				ELSIF stCycleDataNest1.bFail AND stCycleDataNest2.bFail THEN
					
					IF ctuRejectPart.CV > 1 AND NOT bPartPresentNest1 AND NOT bPartPresentNest2 THEN
						
						(* Renan Added 10Jul26 - Puck Locker *)
						IF bPuckLockerEnable THEN
							GVL_Stations.stPuckLocker.nRequestedRelease 		:= USINT#0;
							GVL_Stations.stPuckLocker.bApplyDisposition 		:= TRUE;
						END_IF
						(*\Renan Added 10Jul26 - Puck Locker *)
						
						eCycleState												:= E_General_ProcessCycle.NEST_CLEARING;
					
					ELSIF ctuRejectPart.CV > 1 AND ( bPartPresentNest1 OR bPartPresentNest2) THEN
						
						bRejectPartFault										:= TRUE; 		
					
					END_IF;
					
					sMachineMessage												:= 'REMOVE PART FROM BOTH NESTS AND PUT IN REJECT CHUTE';
					
				END_IF
				
E_General_ProcessCycle.NEST_CLEARING:

				stCamera.CMD.CameraCMD.ContinuousPartPresent1					:= bProcessedPart[0];
				stCamera.CMD.CameraCMD.ContinuousPartPresent2					:= bProcessedPart[1];
				stCamera.CMD.bExecute											:= TRUE;
				
				IF bPuckLockerEnable AND GVL_Stations.stPuckLocker.eState = E_PuckLockerState.WaitingForNestsEmpty THEN
				
					IF (bPartPresentNest1 AND bNest1Flag) OR (bPartPresentNest2 AND bNest2Flag) THEN
						
						sMachineMessage 										:= 'Remove parts from nests to release puck';
						
					ELSE
						
						sMachineMessage 										:= 'Waiting for puck to be released';
						
					END_IF
				
				ELSIF (bPartPresentNest1 AND bNest1Flag) AND NOT (bPartPresentNest2 AND bNest2Flag)  THEN
					
					IF bPuckLockerEnable THEN
						
						sMachineMessage 										:= 'Remove processed part from nest 1 to release puck';
						
					ELSE
						
						sMachineMessage 										:= 'Remove Processed part from nest 1';
						
					END_IF
					
				ELSIF NOT (bPartPresentNest1 AND bNest1Flag) AND (bPartPresentNest2 AND bNest2Flag)  THEN 
					
					IF bPuckLockerEnable THEN
						
						sMachineMessage 										:= 'Remove processed part from nest 2 to release puck';
						
					ELSE
						
						sMachineMessage 										:= 'Remove Processed part from nest 2';
						
					END_IF
					
				ELSIF (bPartPresentNest1 AND bNest1Flag) AND (bPartPresentNest2 AND bNest2Flag) THEN 
					
					IF bPuckLockerEnable THEN
						
						sMachineMessage 										:= 'Remove processed parts to release puck';
						
					ELSE
						
						sMachineMessage 										:= 'Remove Processed parts';
						
					END_IF
					
				ELSIF (NOT bPartPresentNest1 OR NOT bNest1Flag) AND (NOT bPartPresentNest2 OR NOT bNest2Flag)  THEN
					
					sMachineMessage 											:= '';
					eCycleState													:= E_General_ProcessCycle.RESET_ALL_CMD;
									
				END_IF
			
				
END_CASE
END_ACTION

ACTION c_ACT_SaveData:

//SAVING NEST 1 DATA

IF bProcessedPart[0] THEN
		
	IF stCycleDataNest1.bPass THEN
	
		stCycleDataNest1.sGeneralResult			:= 'PASS';

	ELSIF stCycleDataNest1.bFail THEN
	
		stCycleDataNest1.sGeneralResult			:= 'FAIL';

	END_IF

	IF stCycleDataNest1.LSS_Pass THEN
	
		stCycleDataNest1.sHeightTestResult		:= 'PASS';
	
	ELSIF stCycleDataNest1.LSS_Fail THEN
	
		stCycleDataNest1.sHeightTestResult		:= 'FAIL';
	
	END_IF



	IF stCycleDataNest1.LeakTest_Pass THEN
	
		stCycleDataNest1.sLeakTesterResult		:= 'PASS';

	ELSIF stCycleDataNest1.LeakTest_Fail THEN
	
		stCycleDataNest1.sLeakTesterResult		:= 'FAIL';
	
	END_IF
	
	stCycleDataNest1.sDistance1						:= REAL_TO_STRING(stCycleDataNest1.LSS_ScaledHeight[1]);
	stCycleDataNest1.sDistance2						:= REAL_TO_STRING(stCycleDataNest1.LSS_ScaledHeight[2]);
	stCycleDataNest1.sDistance3						:= REAL_TO_STRING(stCycleDataNest1.LSS_ScaledHeight[3]);
	stCycleDataNest1.sDistance4						:= REAL_TO_STRING(stCycleDataNest1.LSS_ScaledHeight[4]);
	
	stCycleDataNest1.sSetpoint1						:= REAL_TO_STRING(nHeightSetPoint);
	stCycleDataNest1.sSetpoint2						:= REAL_TO_STRING(nHeightSetPoint);
	stCycleDataNest1.sSetpoint3						:= REAL_TO_STRING(nHeightSetPoint);
	stCycleDataNest1.sSetpoint4						:= REAL_TO_STRING(nHeightSetPoint);
	
	aDataHistoryNest1[0]						:= stCycleDataNest1;
	
END_IF
	

//SAVING NEST 2 DATA

IF bProcessedPart[1] THEN
	
	IF stCycleDataNest2.bPass THEN
	
		stCycleDataNest2.sGeneralResult			:= 'PASS';

	ELSIF stCycleDataNest2.bFail THEN
	
		stCycleDataNest2.sGeneralResult			:= 'FAIL';

	END_IF

	IF stCycleDataNest2.LSS_Pass THEN
	
		stCycleDataNest2.sHeightTestResult		:= 'PASS';
	
	ELSIF stCycleDataNest2.LSS_Fail THEN
	
		stCycleDataNest2.sHeightTestResult		:= 'FAIL';
	
	END_IF



	IF stCycleDataNest2.LeakTest_Pass THEN
	
		stCycleDataNest2.sLeakTesterResult		:= 'PASS';

	ELSIF stCycleDataNest2.LeakTest_Fail THEN
	
		stCycleDataNest2.sLeakTesterResult		:= 'FAIL';
	
	END_IF
	
	stCycleDataNest2.sDistance1						:= REAL_TO_STRING(stCycleDataNest2.LSS_ScaledHeight[1]);
	stCycleDataNest2.sDistance2						:= REAL_TO_STRING(stCycleDataNest2.LSS_ScaledHeight[2]);
	stCycleDataNest2.sDistance3						:= REAL_TO_STRING(stCycleDataNest2.LSS_ScaledHeight[3]);
	stCycleDataNest2.sDistance4						:= REAL_TO_STRING(stCycleDataNest2.LSS_ScaledHeight[4]);
	
	stCycleDataNest2.sSetpoint1						:= REAL_TO_STRING(nHeightSetPoint);
	stCycleDataNest2.sSetpoint2						:= REAL_TO_STRING(nHeightSetPoint);
	stCycleDataNest2.sSetpoint3						:= REAL_TO_STRING(nHeightSetPoint);
	stCycleDataNest2.sSetpoint4						:= REAL_TO_STRING(nHeightSetPoint);
	
	aDataHistoryNest2[0]						:= stCycleDataNest2;
	
END_IF
END_ACTION

ACTION d_ACT_IO:
//INPUTS

rRejectSensor( CLK := dw_T08_EL1809.iRejectSensor);

bDoorClosingFlag					:= (eCycleState = E_General_ProcessCycle.CLOSE_PROCESS_DOOR) OR (eCycleState = E_General_ProcessCycle.WAIT_CLOSE_PROCESS_DOOR) OR 
										bDoorClosingInitFlag;
bDoorOpeningFlag					:= eCycleState = E_General_ProcessCycle.OPEN_PROCESS_DOOR;

bProcessDoorClosedConditionFlag		:=  eCycleState = E_General_ProcessCycle.EXTEND_PROCESS_CYLINDER OR
										eCycleState = E_General_ProcessCycle.WAIT_EXTEND_PROCESS_CYLINDER OR
										eCycleState = E_General_ProcessCycle.RETRACT_PROCESS_CYLINDER OR
										eCycleState = E_General_ProcessCycle.WAIT_RETRACT_PROCESS_CYLINDER OR
										eCycleState = E_General_ProcessCycle.HOLD_PART OR
										eCycleState = E_General_ProcessCycle.WAIT_HOLD_PART OR
										eCycleState = E_General_ProcessCycle.RELEASE_PART OR
										eCycleState = E_General_ProcessCycle.WAIT_RELEASE_PART OR
										eCycleState = E_General_ProcessCycle.VACUUM_CYLINDER_EXTENSION OR
										eCycleState = E_General_ProcessCycle.WAIT_VACUUM_CYLINDER_EXTENSION OR
										eCycleState = E_General_ProcessCycle.VACUUM_CYLINDER_RETRACTION OR
										eCycleState = E_General_ProcessCycle.WAIT_VACUUM_CYLINDER_RETRACTION;
					

										

										
tonTwoHandsSignal( IN := stTwinSAFE.qTwoHandsSafe , PT := stTimers.tTwoHandsSignal);						
				
bTwoHandsSignal						:= tonTwoHandsSignal.Q;
		
dw_T09_EL2809.qIndicatorLED1_Red	:= stCycleDataNest1.bFail;		
dw_T09_EL2809.qIndicatorLED1_Green	:= stCycleDataNest1.bPass;	
dw_T09_EL2809.qIndicatorLED2_Red	:= stCycleDataNest2.bFail;		
dw_T09_EL2809.qIndicatorLED2_Green	:= stCycleDataNest2.bPass;	

bPartPresent[0]					:= 	bProcessedPart[0];
bPartPresent[1]					:= 	bProcessedPart[1];
	

				
stTwinSAFE.iMachineHoming_Manual		:= 	stMachineStatus.eMachineState = E_MachineState.SAFETY OR
										stMachineStatus.eMachineState = E_MachineState.SYSTEM_INITIALISING OR 
										stMachineStatus.eMachineState = E_MachineState.MANUAL_MODE;												
										
//General Stations CMD
	
stVacuumCylinder.CMD.bAbort			:= bGeneralAbort;
stCamera.CMD.bAbort					:= bGeneralAbort;	
stLeakTesters.CMD.bAbort			:= bGeneralAbort;	
stLSS.CMD.bAbort					:= bGeneralAbort;
stProcessCylinder.CMD.bAbort		:= bGeneralAbort;
stProcessDoor.CMD.bAbort			:= bGeneralAbort;

stVacuumCylinder.CMD.bEnable		:= bGeneralEnable;
stCamera.CMD.bEnable				:= bGeneralEnable;	
stLeakTesters.CMD.bEnable			:= bGeneralEnable;	
stLSS.CMD.bEnable					:= bGeneralEnable;
stProcessCylinder.CMD.bEnable		:= bGeneralEnable;
stProcessDoor.CMD.bEnable			:= bGeneralEnable;

stVacuumCylinder.CMD.bReset			:= bGeneralRST;
stCamera.CMD.bReset					:= bGeneralRST;	
stLeakTesters.CMD.bReset			:= bGeneralRST;	
stLSS.CMD.bReset					:= bGeneralRST;
stProcessCylinder.CMD.bReset		:= bGeneralRST;
stProcessDoor.CMD.bReset			:= bGeneralRST;

stVacuumCylinder.CMD.bManualMode	:= bGeneralManualMode;
stCamera.CMD.bManualMode			:= bGeneralManualMode;
stLeakTesters.CMD.bManualMode		:= bGeneralManualMode;
stLSS.CMD.bManualMode				:= bGeneralManualMode;
stProcessCylinder.CMD.bManualMode	:= bGeneralManualMode;
stProcessDoor.CMD.bManualMode		:= bGeneralManualMode;
END_ACTION

END_PROGRAM

// ---- POUs/B_STATIONS/B_5_PUCK_LOCKER/B_5_1_PRG_PuckLocker.TcPOU
PROGRAM B_5_1_PRG_PuckLocker
VAR
	// ============================================================
    // Local process variables
    // ============================================================
    eMode                       : E_PuckLockerMode;

    bPuckPresentRaw             : BOOL;
    bPuckPresent                : BOOL;

    bPuckSensorsMismatchRaw     : BOOL;
    bPuckSensorsMismatch        : BOOL;

    bEnableEmptyPuckBypass      : BOOL;


    // ============================================================
    // Edge detection
    // ============================================================
    rTrigPuckPresent          : R_TRIG;
    fTrigPuckPresent          : F_TRIG;

    rTrigApplyDisposition     : R_TRIG;
    rTrigEmptyPuckBypass      : R_TRIG;
    rTrigAcknowledgeFault     : R_TRIG;


    // ============================================================
    // Timers
    // ============================================================
    tonPuckPresentOnDelay        : TON;
    tonPuckPresentOffDelay       : TON;

    tonPuckMismatchDelay         : TON;
	tonPuckPresentDebounce		 : TON;
	
    tonPinLockDelay              : TON;
	
END_VAR

// =================================================================
// 1. Engineering / HMI configuration
// =================================================================
// eMode should be persistent through your existing GVL_HMI Persistent
// implementation, or copied there from the Engineering page.
// =================================================================
// Puck locker HMI mode selection
// =================================================================


(* Renan Added 10Jul26 - Puck Locker common code *)


    IF NOT GVL_HMI.bPuckLockerGateEnable THEN
        GVL_HMI.bPuckLockerSkipEnable := FALSE;
    END_IF;

    IF NOT GVL_HMI.bPuckLockerGateEnable THEN

        eMode := E_PuckLockerMode.Disabled;

    ELSIF GVL_HMI.bPuckLockerSkipEnable THEN

        eMode := E_PuckLockerMode.EnabledWithEmptyPuckBypass;

    ELSE

        eMode := E_PuckLockerMode.Enabled;

    END_IF;

    GVL_HMI.ePuckLockerMode := eMode;
    GVL_HMI.stPuckLocker.eMode := eMode;


(*\Renan Added 10Jul26 - Puck Locker common code *)

// Skip option is never allowed while gate is disabled.
IF NOT GVL_HMI.bPuckLockerGateEnable THEN
    GVL_HMI.bPuckLockerSkipEnable := FALSE;
END_IF;

// Convert HMI toggles into the internal locker mode.
IF NOT GVL_HMI.bPuckLockerGateEnable THEN

    eMode := E_PuckLockerMode.Disabled;

ELSIF GVL_HMI.bPuckLockerSkipEnable THEN

    eMode := E_PuckLockerMode.EnabledWithEmptyPuckBypass;

ELSE

    eMode := E_PuckLockerMode.Enabled;

END_IF;

// Keep existing status/interface compatible.
GVL_HMI.ePuckLockerMode := eMode;
GVL_HMI.stPuckLocker.eMode := eMode;


// =================================================================
// 2. Read physical inputs
// =================================================================
GVL_Stations.stPuckLocker.bPuckSensorUp 	:= GVL_IO.dw_T08_EL1809.iPuckSensorUp;
GVL_Stations.stPuckLocker.bPuckSensorDown 	:= GVL_IO.dw_T08_EL1809.iPuckSensorDown;

// =================================================================
// 3. Validate puck presence
// =================================================================
// The puck is considered correctly positioned only when both sensors
// are active simultaneously.
bPuckPresentRaw := GVL_Stations.stPuckLocker.bPuckSensorUp AND GVL_Stations.stPuckLocker.bPuckSensorDown;

GVL_IO.stTwinSAFE.iPuckError := GVL_Stations.stPuckLocker.bUnexpectedRemovalFault;

// One sensor ON and the other OFF may be caused by:
// - puck moving through the sensing area;
// - puck not aligned;
// - puck partially lifted;
// - sensor issue.
bPuckSensorsMismatchRaw :=GVL_Stations.stPuckLocker.bPuckSensorUp XOR GVL_Stations.stPuckLocker.bPuckSensorDown;

// Require both sensors active for 100 ms before confirming puck.
tonPuckPresentOnDelay(IN := bPuckPresentRaw,PT := T#100MS);

// Require both sensors inactive for 100 ms before confirming absence.
tonPuckPresentOffDelay(IN := NOT bPuckPresentRaw,PT := T#100MS);


IF tonPuckPresentOnDelay.Q THEN

    bPuckPresent := TRUE;

ELSIF tonPuckPresentOffDelay.Q THEN

    bPuckPresent := FALSE;

END_IF

// Debounce puck present
tonPuckPresentDebounce(IN := bPuckPresentRaw, PT := T#100MS);

// Debounced puck detection
GVL_Stations.stPuckLocker.bPuckDetected := tonPuckPresentDebounce.Q;

// Keep mismatch indication only after a short delay, so normal puck
// movement does not generate false warnings.
tonPuckMismatchDelay(IN := bPuckSensorsMismatchRaw,PT := T#500MS);

bPuckSensorsMismatch := tonPuckMismatchDelay.Q;

// =================================================================
// 4. Edge detection
// =================================================================
rTrigPuckPresent(CLK := bPuckPresent);

fTrigPuckPresent(CLK := bPuckPresent);

rTrigApplyDisposition(CLK := GVL_Stations.stPuckLocker.bApplyDisposition);

rTrigEmptyPuckBypass(CLK := GVL_HMI.stPuckLocker.bCmdEmptyPuckBypass);

rTrigAcknowledgeFault(CLK := GVL_HMI.stPuckLocker.bCmdAcknowledgeRemovalFault);


// =================================================================
// 5. Latch disposition request from MachineCtrl
// =================================================================
// MachineCtrl should write these values once, after both final nest
// results are known:
//
// PASS / PASS:
// nRequestedRelease := 2;
// nRequestedRemoval := 0;
//
// PASS / FAIL or FAIL / PASS:
// nRequestedRelease := 1;
// nRequestedRemoval := 0;
//
// FAIL / FAIL:
// nRequestedRelease := 0;
// nRequestedRemoval := 1;
//
// bApplyDisposition := TRUE;
IF rTrigApplyDisposition.Q THEN

    IF GVL_Stations.stPuckLocker.nRequestedRelease > USINT#2 THEN
        GVL_Stations.stPuckLocker.nPucksAllowedToPass := USINT#2;
    ELSE
        GVL_Stations.stPuckLocker.nPucksAllowedToPass :=
            GVL_Stations.stPuckLocker.nRequestedRelease;
    END_IF

    GVL_Stations.stPuckLocker.bDispositionPending := TRUE;
    GVL_Stations.stPuckLocker.bApplyDisposition := FALSE;

END_IF


// =================================================================
// 6. Default values
// =================================================================
GVL_Stations.stPuckLocker.bRemovalAllowed := FALSE;
bEnableEmptyPuckBypass := FALSE;

tonPinLockDelay(IN := GVL_Stations.stPuckLocker.eState = E_PuckLockerState.LockingPuck AND bPuckPresent, PT := T#300MS);

IF stMachineStatus.bInitialising OR stMachineStatus.eMachineState = E_MachineState.SYSTEM_INITIALISING THEN

    f_ACT_ResetPuckLocker();
    RETURN;

END_IF

// =================================================================
// 8. Main Puck Locker State Machine
// =================================================================
CASE GVL_Stations.stPuckLocker.eState OF


    // ------------------------------------------------------------
    // Locker disabled.
    // Pin remains down and does not interfere with puck movement.
    // ------------------------------------------------------------
    E_PuckLockerState.Disabled:

        GVL_Stations.stPuckLocker.bPinCommandUp := FALSE;

        GVL_Stations.stPuckLocker.bPuckLocked := FALSE;
        GVL_Stations.stPuckLocker.bUnexpectedRemovalFault := FALSE;

        GVL_Stations.stPuckLocker.nPucksAllowedToPass := 0;
        GVL_Stations.stPuckLocker.nPucksToRemove := 0;

        GVL_Stations.stPuckLocker.bDispositionPending := FALSE;
        GVL_Stations.stPuckLocker.bDispositionHandled := FALSE;

        IF eMode <> E_PuckLockerMode.Disabled THEN

            GVL_Stations.stPuckLocker.eState := E_PuckLockerState.WaitingForPuck;

        END_IF


    // ------------------------------------------------------------
    // Pin remains down. Wait for a properly centred puck.
    // ------------------------------------------------------------
    E_PuckLockerState.WaitingForPuck:

        GVL_Stations.stPuckLocker.bPinCommandUp := FALSE;
        GVL_Stations.stPuckLocker.bPuckLocked := FALSE;

        IF eMode = E_PuckLockerMode.Disabled THEN

            GVL_Stations.stPuckLocker.eState := E_PuckLockerState.Disabled;

        ELSIF bPuckPresent
              AND GVL_Stations.stPuckLocker.nPucksAllowedToPass = 0
              AND GVL_Stations.stPuckLocker.nPucksToRemove = 0 THEN

            GVL_Stations.stPuckLocker.eState := E_PuckLockerState.LockingPuck;

        END_IF


    // ------------------------------------------------------------
    // Pin command is up.
    // No physical feedback exists, so locking is accepted after
    // 300 ms while the puck stays detected.
    // ------------------------------------------------------------
    E_PuckLockerState.LockingPuck:

        GVL_Stations.stPuckLocker.bPinCommandUp := TRUE;
		GVL_Stations.stPuckLocker.bPuckLocked := FALSE;
	
		IF eMode = E_PuckLockerMode.Disabled THEN
	
			GVL_Stations.stPuckLocker.eState := E_PuckLockerState.Disabled;
	
		ELSIF NOT bPuckPresent THEN
	
			// Puck was not fully captured yet.
			// Return to waiting state without fault.
			GVL_Stations.stPuckLocker.eState := E_PuckLockerState.WaitingForPuck;
	
		ELSIF tonPinLockDelay.Q THEN
	
			GVL_Stations.stPuckLocker.bPuckLocked := TRUE;
			GVL_Stations.stPuckLocker.eState := E_PuckLockerState.Locked;
	
		END_IF


    // ------------------------------------------------------------
    // Puck captured by locker pin.
    // Wait for process disposition, bypass request or fault.
    // ------------------------------------------------------------
    E_PuckLockerState.Locked:

        GVL_Stations.stPuckLocker.bPinCommandUp := TRUE;
        GVL_Stations.stPuckLocker.bPuckLocked := TRUE;


        // Bypass is only allowed in the configured bypass mode.
        // It is disabled once a process disposition is pending.
        bEnableEmptyPuckBypass := (eMode = E_PuckLockerMode.EnabledWithEmptyPuckBypass) AND NOT GVL_Stations.stPuckLocker.bDispositionPending AND NOT GVL_Stations.stPuckLocker.bUnexpectedRemovalFault;


        // Puck disappeared while pin should have been holding it.
        IF NOT bPuckPresent THEN

            GVL_Stations.stPuckLocker.bUnexpectedRemovalFault := TRUE;
            GVL_Stations.stPuckLocker.eState := E_PuckLockerState.UnexpectedPuckRemovalFault;


        // Empty puck bypass confirmed through HMI.
        ELSIF rTrigEmptyPuckBypass.Q
              AND bEnableEmptyPuckBypass THEN

            GVL_Stations.stPuckLocker.nPucksAllowedToPass := 1;
            GVL_Stations.stPuckLocker.nPucksToRemove := 0;

            GVL_HMI.stPuckLocker.bCmdEmptyPuckBypass := FALSE;

            GVL_Stations.stPuckLocker.eState := E_PuckLockerState.ReleasingPucks;


        // Final disposition received from MachineCtrl.
		ELSIF GVL_Stations.stPuckLocker.bDispositionPending THEN

			GVL_Stations.stPuckLocker.bDispositionPending := FALSE;
		
			// Release is authorised, but the pin must remain up until
			// both nests are empty. This ensures the PASS part was placed
			// back onto the locked puck before it can be released.
			IF GVL_Stations.stPuckLocker.nPucksAllowedToPass > 0 THEN
		
				GVL_Stations.stPuckLocker.eState := E_PuckLockerState.WaitingForNestsEmpty;
		
			END_IF
		END_IF


    E_PuckLockerState.WaitingForNestsEmpty:

		// Keep puck physically locked while either nest still contains
		// a product.
		GVL_Stations.stPuckLocker.bPinCommandUp := TRUE;
		GVL_Stations.stPuckLocker.bPuckLocked := TRUE;
	
		IF NOT bPuckPresent THEN
	
			GVL_Stations.stPuckLocker.bUnexpectedRemovalFault := TRUE;
	
			GVL_Stations.stPuckLocker.eState := E_PuckLockerState.UnexpectedPuckRemovalFault;
	
		ELSIF GVL_Stations.stPuckLocker.bNestsEmpty AND GVL_Stations.stPuckLocker.nPucksAllowedToPass > 0 THEN
	
			GVL_Stations.stPuckLocker.eState := E_PuckLockerState.ReleasingPucks;
	
		END_IF
		
    // ------------------------------------------------------------
    // Pin is down. One or two authorised pucks may pass.
    // A puck is counted when it clears both sensors.
    // ------------------------------------------------------------
    E_PuckLockerState.ReleasingPucks:

        GVL_Stations.stPuckLocker.bPinCommandUp := FALSE;
        GVL_Stations.stPuckLocker.bPuckLocked := FALSE;

        IF fTrigPuckPresent.Q
           AND GVL_Stations.stPuckLocker.nPucksAllowedToPass > 0 THEN

            GVL_Stations.stPuckLocker.nPucksAllowedToPass := GVL_Stations.stPuckLocker.nPucksAllowedToPass - 1;

        END_IF

        // All authorised pucks passed through the locker.
		// Return to rest/waiting state. No timeout is required here.
		IF GVL_Stations.stPuckLocker.nPucksAllowedToPass = 0
		AND NOT bPuckPresent THEN
		
			GVL_Stations.stPuckLocker.eState := E_PuckLockerState.WaitingForPuck;
		
		END_IF


    // ------------------------------------------------------------
    // Puck was removed unexpectedly while locked.
    // Pin stays down for safe recovery.
    //
    // Operator must return the puck to the sensor area and an
    // authorised user must acknowledge the event.
    // ------------------------------------------------------------
    E_PuckLockerState.UnexpectedPuckRemovalFault:

		GVL_Stations.stPuckLocker.bPinCommandUp := TRUE;
		GVL_Stations.stPuckLocker.bPuckLocked := FALSE;
	
		GVL_Stations.stPuckLocker.bUnexpectedRemovalFault := TRUE;
	
		IF eMode = E_PuckLockerMode.Disabled THEN
	
			GVL_Stations.stPuckLocker.eState := E_PuckLockerState.Disabled;
	
		ELSIF bPuckPresent AND rTrigAcknowledgeFault.Q THEN
		
			GVL_HMI.stPuckLocker.bCmdAcknowledgeRemovalFault := FALSE;
			GVL_Stations.stPuckLocker.bUnexpectedRemovalFault := FALSE;
			GVL_Stations.stPuckLocker.eState := E_PuckLockerState.LockingPuck;

		END_IF

END_CASE


// =================================================================
// 8. Write HMI interface
// =================================================================
GVL_HMI.stPuckLocker.bEnableEmptyPuckBypass := bEnableEmptyPuckBypass;

GVL_HMI.stPuckLocker.bPuckDetected := bPuckPresent;

GVL_HMI.stPuckLocker.bPuckLocked := GVL_Stations.stPuckLocker.bPuckLocked;

GVL_HMI.stPuckLocker.bPuckSensorMismatch := bPuckSensorsMismatch;

GVL_HMI.stPuckLocker.bUnexpectedRemovalFault := GVL_Stations.stPuckLocker.bUnexpectedRemovalFault;

GVL_HMI.stPuckLocker.bShowUnexpectedRemovalPopup := GVL_Stations.stPuckLocker.bUnexpectedRemovalFault;

GVL_HMI.stPuckLocker.nPucksAllowedToPass := GVL_Stations.stPuckLocker.nPucksAllowedToPass;


// This can remain FALSE if the HMI itself opens the confirmation
// popup after the operator presses the bypass button.
GVL_HMI.stPuckLocker.bShowEmptyPuckPopup := FALSE;



GVL_HMI.stPuckLocker.sMessage := GVL_Stations.stPuckLocker.sMessage;

// =================================================================
// 10. Physical output
// =================================================================
// This PRG must remain the only writer of the locker output.
GVL_IO.dw_T09_EL2809.qPuckLockerPinCommand := NOT GVL_Stations.stPuckLocker.bPinCommandUp;

ACTION f_ACT_ResetPuckLocker:
// ================================================================
// f_ACT_ResetPuckLocker
//
// Safe reset of puck locker internal state.
// Pin is commanded to release position.
// ================================================================

GVL_Stations.stPuckLocker.eState := E_PuckLockerState.WaitingForPuck;

GVL_Stations.stPuckLocker.bPinCommandUp := FALSE;
GVL_Stations.stPuckLocker.bPuckLocked := FALSE;
GVL_Stations.stPuckLocker.bRemovalAllowed := FALSE;

GVL_Stations.stPuckLocker.bUnexpectedRemovalFault := FALSE;

GVL_Stations.stPuckLocker.nPucksAllowedToPass := 0;
GVL_Stations.stPuckLocker.nPucksToRemove := 0;

GVL_Stations.stPuckLocker.nRequestedRelease := 0;
GVL_Stations.stPuckLocker.nRequestedRemoval := 0;

GVL_Stations.stPuckLocker.bApplyDisposition := FALSE;
GVL_Stations.stPuckLocker.bDispositionPending := FALSE;
GVL_Stations.stPuckLocker.bDispositionHandled := FALSE;

GVL_HMI.stPuckLocker.bCmdEmptyPuckBypass := FALSE;
GVL_HMI.stPuckLocker.bCmdAcknowledgeRemovalFault := FALSE;

GVL_HMI.stPuckLocker.bEnableEmptyPuckBypass := FALSE;
GVL_HMI.stPuckLocker.bShowUnexpectedRemovalPopup := FALSE;
GVL_HMI.stPuckLocker.bShowEmptyPuckPopup := FALSE;

GVL_HMI.stPuckLocker.bUnexpectedRemovalFault := FALSE;
GVL_HMI.stPuckLocker.nPucksAllowedToPass := 0;
GVL_HMI.stPuckLocker.sMessage := '';
END_ACTION

END_PROGRAM

// ---- POUs/D_CSV/D_1_PRG_CycleDataCSV.TcPOU
PROGRAM D_1_PRG_CycleDataCSV
VAR_INPUT
	
	stCycleDataNest1		: ST_CycleData;
	stCycleDataNest2		: ST_CycleData;
	bWriteNest1				: BOOL;
	bWriteNest2				: BOOL;
	
	
END_VAR
VAR_OUTPUT
	
	bCSVDone				: BOOL;
	bReady					: BOOL;
	
END_VAR
VAR
	sFileName		: T_MaxString := 'C:\Temp\USW_STN13_#date#.csv';(* CSV destination file path and name *)
	sCSVLine		: T_MaxString := '#1#;#2#;#3#;#4#;#5#;#6#;#7#;#8#;#9#,#10#,#11#,#12#,#13,#14,#15,#16,#17,#18#$L';
	bBusy			: BOOL;
	bError			: BOOL;
	nErrId			: UDINT;
	hFile			: UINT		:= 0;
	step			: DWORD 	:= 0;
	fbFileOpen		: FB_FileOpen;(* Opens file *)
	fbFileClose		: FB_FileClose;(* Closes file *)
	fbFilePuts		: FB_FilePuts;(* Writes one record (line) *)
	
	done: BOOL;
	
	f1_Nest			: STRING;
	f2_GeneralResult: STRING;
	f3_HeightResult	: STRING;
	f4_LeakTesterResult	: STRING;
	f5_Distance1	: STRING;
	f6_Distance2	: STRING;
	f7_Distance3	: STRING;
	f8_Distance4	: STRING;
	f9_Setpoint1	: STRING;
	f10_Setpoint2	: STRING;
	f11_Setpoint3	: STRING;
	f12_Setpoint4	: STRING;
	f13_RawValue1	: STRING;
	f14_RawValue2	: STRING;
	f15_RawValue3	: STRING;
	f16_RawValue4	: STRING;
	f17_Date		: STRING;
	f18_Time		: STRING;
	
	bWritingFirstRow : BOOL;
	bWrite			: BOOL;
	rWriteNest1		: R_TRIG;
	rWriteNest2		: R_TRIG;
	
	rError			: R_TRIG;
	
END_VAR



IF 	step = 0 THEN
	
		bReady		:= TRUE;

ELSE 	bReady		:= FALSE;
END_IF

CASE step OF
	0:	(* Wait for rising edge at bWrite variable *)
		bCSVDone	:= FALSE;
		IF bWrite	 THEN
			
			bWrite	:= FALSE;
			bBusy 	:= TRUE;
			bError	:= FALSE;
			nErrId	:= 0;
			hFile	:= 0;
			step 	:= 1;
			
		END_IF
		
	1:	(* Open source file *)
		fbFileOpen(  bExecute := FALSE  );
		fbFileOpen( sNetId := NetAmsIdLocal, 
					sPathName := sFileName, 
					nMode := FOPEN_MODEAPPEND OR FOPEN_MODETEXT,
					ePath := PATH_GENERIC, 
					bExecute := TRUE );
		step := 2;
	
	2:(* Wait until open not busy *)
		fbFileOpen( bExecute := FALSE, bError => bError, nErrID => nErrID, hFile => hFile );
		IF NOT fbFileOpen.bBusy THEN
			IF NOT fbFileOpen.bError THEN
				step := 3;
			ELSE(* Error: file not found? *)
				step := 100;
			END_IF
		END_IF

	3:(* Convert one PLC record to CSV format *)
		
		FindAndReplace(pSrcString:= ADR(sCSVLine), pDeleteString:= ADR('#1#'), pInsertString:= ADR(f1_Nest), pDstString:= ADR(sCSVLine), nDstSize:= SIZEOF(sCSVLine));
		FindAndReplace(pSrcString:= ADR(sCSVLine), pDeleteString:= ADR('#2#'), pInsertString:= ADR(f2_GeneralResult), pDstString:= ADR(sCSVLine), nDstSize:= SIZEOF(sCSVLine));
		FindAndReplace(pSrcString:= ADR(sCSVLine), pDeleteString:= ADR('#3#'), pInsertString:= ADR(f3_HeightResult), pDstString:= ADR(sCSVLine), nDstSize:= SIZEOF(sCSVLine));
		FindAndReplace(pSrcString:= ADR(sCSVLine), pDeleteString:= ADR('#4#'), pInsertString:= ADR(f4_LeakTesterResult), pDstString:= ADR(sCSVLine), nDstSize:= SIZEOF(sCSVLine));
		FindAndReplace(pSrcString:= ADR(sCSVLine), pDeleteString:= ADR('#5#'), pInsertString:= ADR(f5_Distance1), pDstString:= ADR(sCSVLine), nDstSize:= SIZEOF(sCSVLine));
		FindAndReplace(pSrcString:= ADR(sCSVLine), pDeleteString:= ADR('#6#'), pInsertString:= ADR(f6_Distance2), pDstString:= ADR(sCSVLine), nDstSize:= SIZEOF(sCSVLine));
		FindAndReplace(pSrcString:= ADR(sCSVLine), pDeleteString:= ADR('#7#'), pInsertString:= ADR(f7_Distance3), pDstString:= ADR(sCSVLine), nDstSize:= SIZEOF(sCSVLine));
		FindAndReplace(pSrcString:= ADR(sCSVLine), pDeleteString:= ADR('#8#'), pInsertString:= ADR(f8_Distance4), pDstString:= ADR(sCSVLine), nDstSize:= SIZEOF(sCSVLine));
		FindAndReplace(pSrcString:= ADR(sCSVLine), pDeleteString:= ADR('#9#'), pInsertString:= ADR(f9_Setpoint1), pDstString:= ADR(sCSVLine), nDstSize:= SIZEOF(sCSVLine));
		FindAndReplace(pSrcString:= ADR(sCSVLine), pDeleteString:= ADR('#10#'), pInsertString:= ADR(f10_Setpoint2), pDstString:= ADR(sCSVLine), nDstSize:= SIZEOF(sCSVLine));
		FindAndReplace(pSrcString:= ADR(sCSVLine), pDeleteString:= ADR('#11#'), pInsertString:= ADR(f11_Setpoint3), pDstString:= ADR(sCSVLine), nDstSize:= SIZEOF(sCSVLine));
		FindAndReplace(pSrcString:= ADR(sCSVLine), pDeleteString:= ADR('#12#'), pInsertString:= ADR(f12_Setpoint4), pDstString:= ADR(sCSVLine), nDstSize:= SIZEOF(sCSVLine));
		FindAndReplace(pSrcString:= ADR(sCSVLine), pDeleteString:= ADR('#13#'), pInsertString:= ADR(f13_RawValue1), pDstString:= ADR(sCSVLine), nDstSize:= SIZEOF(sCSVLine));
		FindAndReplace(pSrcString:= ADR(sCSVLine), pDeleteString:= ADR('#14#'), pInsertString:= ADR(f14_RawValue2), pDstString:= ADR(sCSVLine), nDstSize:= SIZEOF(sCSVLine));
		FindAndReplace(pSrcString:= ADR(sCSVLine), pDeleteString:= ADR('#15#'), pInsertString:= ADR(f15_RawValue3), pDstString:= ADR(sCSVLine), nDstSize:= SIZEOF(sCSVLine));
		FindAndReplace(pSrcString:= ADR(sCSVLine), pDeleteString:= ADR('#16#'), pInsertString:= ADR(f16_RawValue4), pDstString:= ADR(sCSVLine), nDstSize:= SIZEOF(sCSVLine));	
		FindAndReplace(pSrcString:= ADR(sCSVLine), pDeleteString:= ADR('#17#'), pInsertString:= ADR(f17_Date), pDstString:= ADR(sCSVLine), nDstSize:= SIZEOF(sCSVLine));
		FindAndReplace(pSrcString:= ADR(sCSVLine), pDeleteString:= ADR('#18#'), pInsertString:= ADR(f18_Time), pDstString:= ADR(sCSVLine), nDstSize:= SIZEOF(sCSVLine));
		done:=TRUE;
		
		IF done THEN
			step := 4;
			done := FALSE;
		ELSE
			step := 3;
		END_IF
		
		
	4:	(* Write single text line *)
		fbFilePuts( bExecute := FALSE );
		fbFilePuts( sNetId := '', 
					hFile := hFile, 
					sLine := sCSVLine, 
					bExecute := TRUE );
		step := 5;

	5:(* Wait until write not busy *)
		fbFilePuts( bExecute := FALSE, bError => bError, nErrID => nErrID );
		IF NOT fbFilePuts.bBusy THEN
			IF NOT fbFilePuts.bError THEN
				step := 10;
			ELSE(* Error *)
				step := 100;
			END_IF
		END_IF

	10:	(* Close source file *)
		fbFileClose( bExecute := FALSE );
		fbFileClose( sNetId := '', hFile := hFile, bExecute := TRUE );
		sCSVLine:= '#1#;#2#;#3#;#4#;#5#;#6#;#7#;#8#;#9#,#10#,#11#,#12#,#13#,#14#,#15#,#16#,#17#$L';
		step := 11;

	11:(* Wait until close not busy *)
		fbFileClose( bExecute := FALSE, bError => bError, nErrID => nErrID );
		IF ( NOT fbFileClose.bBusy ) THEN
			bWritingFirstRow	:= FALSE;
			
			hFile := 0;
			step := 100;
		END_IF

	100: (* Error or ready step => cleanup *)
		IF ( hFile <> 0 ) THEN
			step := 10; (* Close the source file *)
		ELSE
			bBusy := FALSE;
			step := 0;	(* Ready *)
			bCSVDone	:= TRUE;
		END_IF

END_CASE

IF (lastDateCSV <> sSystemDate) AND NOT (dw_T04_EL1918.iResetButton	OR stTester.bReset) THEN
lastDateCSV:= sSystemDate;
sFileName:= 'C:\Users\Administrator\Desktop\csv\CycleData_#date#.csv';
FindAndReplace(pSrcString:= ADR(sFileName), pDeleteString:= ADR('#date#'), pInsertString:= ADR(lastDateCSV), pDstString:= ADR(sFileName), nDstSize:= SIZEOF(sFileName));

f1_Nest			:= 'NEST';
f2_GeneralResult:= 'GENERAL RESULTS';
f3_HeightResult	:= 'HEIGHT CHECK RESULTS';
f4_LeakTesterResult	:= 'LEAK TESTER RESULTS';
f5_Distance1	:= 'DISTANCE 1';
f6_Distance2	:= 'DISTANCE 2';
f7_Distance3	:= 'DISTANCE 3';
f8_Distance4	:= 'DISTANCE 4';
f9_Setpoint1	:= 'SETPOINT 1';
f10_Setpoint2	:= 'SETPOINT 2';
f11_Setpoint3	:= 'SETPOINT 3';
f12_Setpoint4	:= 'SETPOINT 4';
f13_RawValue1	:= 'RAW HEIGHT 1';
f14_RawValue2	:= 'RAW HEIGHT 2';
f15_RawValue3	:= 'RAW HEIGHT 3';
f16_RawValue4	:= 'RAW HEIGHT 4';
f17_Date		:= 'DATE';
f18_Time		:= 'TIME';
bWrite			:= TRUE;
bWritingFirstRow	:= TRUE;

END_IF

IF NOT bWritingFirstRow THEN
	ACT_LinkingVariables();
END_IF

rError(CLK := bError);

bCSVError		:= rError.Q;

IF bWritingFirstRow AND (dw_T04_EL1918.iResetButton OR stTester.bReset) THEN
	
	lastDateCSV			:= '0';
	bCSVError			:= FALSE;			

END_IF

ACTION ACT_LinkingVariables:
rWriteNest1( CLK := bWriteNest1);
rWriteNest2( CLK := bWriteNest2);

IF rWriteNest1.Q THEN
	
	f1_Nest			:= INT_TO_STRING(stCycleDataNest1.nNest);
	f2_GeneralResult:= stCycleDataNest1.sGeneralResult;
	f3_HeightResult	:= stCycleDataNest1.sHeightTestResult;
	f4_LeakTesterResult	:= stCycleDataNest1.sLeakTesterResult;
	f5_Distance1	:= stCycleDataNest1.sDistance1;
	f6_Distance2	:= stCycleDataNest1.sDistance2;
	f7_Distance3	:= stCycleDataNest1.sDistance3;
	f8_Distance4	:= stCycleDataNest1.sDistance4;
	f9_Setpoint1	:= stCycleDataNest1.sSetpoint1;
	f10_Setpoint2	:= stCycleDataNest1.sSetpoint2;
	f11_Setpoint3	:= stCycleDataNest1.sSetpoint3;
	f12_Setpoint4	:= stCycleDataNest1.sSetpoint4;
	f13_RawValue1	:= REAL_TO_STRING(stCycleDataNest1.LSS_anRawMeasurement[1]);
	f14_RawValue2	:= REAL_TO_STRING(stCycleDataNest1.LSS_anRawMeasurement[2]);
	f15_RawValue3	:= REAL_TO_STRING(stCycleDataNest1.LSS_anRawMeasurement[3]);
	f16_RawValue4	:= REAL_TO_STRING(stCycleDataNest1.LSS_anRawMeasurement[4]);
	f17_Date		:= stCycleDataNest1.sDate;
	f18_Time		:= stCycleDataNest1.sTime;
	
	bWrite			:= TRUE;

ELSIF rWriteNest2.Q THEN
	
	f1_Nest			:= INT_TO_STRING(stCycleDataNest2.nNest);
	f2_GeneralResult:= stCycleDataNest2.sGeneralResult;
	f3_HeightResult	:= stCycleDataNest2.sHeightTestResult;
	f4_LeakTesterResult	:= stCycleDataNest2.sLeakTesterResult;
	f5_Distance1	:= stCycleDataNest2.sDistance1;
	f6_Distance2	:= stCycleDataNest2.sDistance2;
	f7_Distance3	:= stCycleDataNest2.sDistance3;
	f8_Distance4	:= stCycleDataNest2.sDistance4;
	f9_Setpoint1	:= stCycleDataNest2.sSetpoint1;
	f10_Setpoint2	:= stCycleDataNest2.sSetpoint2;
	f11_Setpoint3	:= stCycleDataNest2.sSetpoint3;
	f12_Setpoint4	:= stCycleDataNest2.sSetpoint4;
	f13_RawValue1	:= REAL_TO_STRING(stCycleDataNest2.LSS_anRawMeasurement[1]);
	f14_RawValue2	:= REAL_TO_STRING(stCycleDataNest2.LSS_anRawMeasurement[2]);
	f15_RawValue3	:= REAL_TO_STRING(stCycleDataNest2.LSS_anRawMeasurement[3]);
	f16_RawValue4	:= REAL_TO_STRING(stCycleDataNest2.LSS_anRawMeasurement[4]);
	f17_Date		:= stCycleDataNest2.sDate;
	f18_Time		:= stCycleDataNest2.sTime;
	
	bWrite			:= TRUE;
	
END_IF
END_ACTION

END_PROGRAM
